(* PLC project bottling_line, Dassault Systèmes ControlBuild 2020 *)
(* stored: creationDateTime 2019-04-23T11:17:34-01:00 *)

CONFIGURATION bottling_line
  VAR_GLOBAL
    generalPanel/acknowledgePB AT 10 : BOOL := false;
    generalPanel/powerUpPB AT 6 : BOOL := false;
    generalPanel/emergencyStopPB AT 7 : BOOL := false;
    generalPanel/manual AT 8 : BOOL := false;
    generalPanel/auto AT 9 : BOOL := false;
    generalPanel/startCyclePB AT 17 : BOOL := false;
    generalPanel/initPB AT 18 : BOOL := false;
    generalPanel/preparationPB AT 19 : BOOL := false;
    generalPanel/productionPB AT 20 : BOOL := false;
    generalPanel/closingPB AT 21 : BOOL := false;
    generalPanel/acknowledgePB/PB AT 10 : BOOL := false;
    generalPanel/acknowledgePB/action AT 39 : BOOL := false;
    generalPanel/acknowledgePB/timeCounter AT 24 : REAL := 0.0;
    generalPanel/acknowledgePB/pulseDuration AT 25 : REAL := 5.0;
    generalPanel/acknowledgePB/PBLogic AT 40 : BOOL := true;
    generalPanel/powerUpPB/PB AT 6 : BOOL := false;
    generalPanel/powerUpPB/action AT 41 : BOOL := false;
    generalPanel/powerUpPB/timeCounter AT 26 : REAL := 0.0;
    generalPanel/powerUpPB/pulseDuration AT 27 : REAL := 5.0;
    generalPanel/powerUpPB/PBLogic AT 42 : BOOL := true;
    generalPanel/emergencyStopPB/pb AT 7 : BOOL := false;
    generalPanel/emergencyStopPB/action AT 43 : BOOL := false;
    generalPanel/emergencyStopPB/PBLogic AT 44 : BOOL := false;
    generalPanel/modesSwitch/leftVariable AT 9 : BOOL := true;
    generalPanel/modesSwitch/rightVariable AT 8 : BOOL := false;
    generalPanel/modesSwitch/leftPosition AT 45 : BOOL := false;
    generalPanel/modesSwitch/rightPosition AT 46 : BOOL := false;
    generalPanel/startCyclePB/PB AT 17 : BOOL := false;
    generalPanel/startCyclePB/action AT 47 : BOOL := false;
    generalPanel/startCyclePB/timeCounter AT 28 : REAL := 0.0;
    generalPanel/startCyclePB/pulseDuration AT 29 : REAL := 5.0;
    generalPanel/startCyclePB/PBLogic AT 48 : BOOL := true;
    generalPanel/initPB/PB AT 18 : BOOL := false;
    generalPanel/initPB/action AT 49 : BOOL := false;
    generalPanel/initPB/timeCounter AT 30 : REAL := 0.0;
    generalPanel/initPB/pulseDuration AT 31 : REAL := 5.0;
    generalPanel/initPB/PBLogic AT 50 : BOOL := true;
    generalPanel/productionSwitch/leftVariable AT 19 : BOOL := true;
    generalPanel/productionSwitch/rightVariable AT 20 : BOOL := false;
    generalPanel/productionSwitch/leftPosition AT 51 : BOOL := false;
    generalPanel/productionSwitch/rightPosition AT 52 : BOOL := false;
    generalPanel/closingPB/PB AT 21 : BOOL := false;
    generalPanel/closingPB/action AT 53 : BOOL := false;
    generalPanel/closingPB/timeCounter AT 32 : REAL := 0.0;
    generalPanel/closingPB/pulseDuration AT 33 : REAL := 5.0;
    generalPanel/closingPB/PBLogic AT 54 : BOOL := true;
    workingModes/powerUpPB AT 6 : BOOL := false;
    workingModes/emergencyStopPB AT 7 : BOOL := false;
    workingModes/manual AT 8 : BOOL := false;
    workingModes/auto AT 9 : BOOL := false;
    workingModes/acknowledgePB AT 10 : BOOL := false;
    workingModes/powerUp AT 5 : BOOL := false;
    workingModes/autoMode AT 28 : BOOL := false;
    workingModes/manualMode AT 29 : BOOL := false;
    workingModes/emStp AT 55 : BOOL := false;
    process/highLevel1 AT 11 : BOOL := false;
    process/lowLevel1 AT 12 : BOOL := false;
    process/highLevel2 AT 13 : BOOL := false;
    process/lowLevel2 AT 14 : BOOL := false;
    process/highLevel3 AT 15 : BOOL := false;
    process/lowLevel3 AT 16 : BOOL := false;
    process/startCyclePB AT 17 : BOOL := false;
    process/initPB AT 18 : BOOL := false;
    process/preparationPB AT 19 : BOOL := false;
    process/productionPB AT 20 : BOOL := false;
    process/closingPB AT 21 : BOOL := false;
    process/pulseGenerator AT 22 : BOOL := false;
    process/bottleFilled AT 23 : BOOL := false;
    process/bottlePresent AT 24 : BOOL := false;
    process/load AT 36 : BOOL := false;
    process/evacuate AT 37 : BOOL := false;
    process/convoy AT 38 : BOOL := false;
    process/pump1 AT 27 : BOOL := false;
    process/pump2 AT 32 : BOOL := false;
    process/valve1 AT 25 : BOOL := false;
    process/valve2 AT 30 : BOOL := false;
    process/valve3 AT 26 : BOOL := false;
    process/valve4 AT 31 : BOOL := false;
    process/loSpeedAgitator AT 35 : BOOL := false;
    process/hiSpeedAgitator AT 34 : BOOL := false;
    process/valve5 AT 33 : BOOL := false;
    process/master/startCyclePB AT 17 : BOOL := false;
    process/master/initPB AT 18 : BOOL := false;
    process/master/preparationPB AT 19 : BOOL := false;
    process/master/productionPB AT 20 : BOOL := false;
    process/master/closingPB AT 21 : BOOL := false;
    process/master/initEnd AT 60 : BOOL := false;
    process/master/preparationEnd AT 61 : BOOL := false;
    process/master/closingEnd AT 62 : BOOL := false;
    process/master/lowLevel3 AT 16 : BOOL := false;
    process/master/initializationRqst AT 59 : BOOL := false;
    process/master/preparationRqst AT 66 : BOOL := false;
    process/master/productionRqst AT 63 : BOOL := false;
    process/master/closingRqst AT 64 : BOOL := false;
    process/master/masterInStandBy AT 65 : BOOL := false;
    process/master/productionWaiting AT 67 : BOOL := false;
    process/master/_X_10 AT 84 : BOOL := true;
    process/master/_X_11 AT 85 : BOOL := false;
    process/master/_X_12 AT 83 : BOOL := false;
    process/master/_X_13 AT 86 : BOOL := false;
    process/master/_X_16 AT 89 : BOOL := false;
    process/master/_X_14 AT 87 : BOOL := false;
    process/master/_X_15 AT 88 : BOOL := false;
    process/tanks/productionRequest AT 63 : BOOL := false;
    process/tanks/closingRequest AT 64 : BOOL := false;
    process/tanks/masterInStandBy AT 65 : BOOL := false;
    process/tanks/highLevel1 AT 11 : BOOL := false;
    process/tanks/highLevel2 AT 13 : BOOL := false;
    process/tanks/highLevel3 AT 15 : BOOL := false;
    process/tanks/lowLevel1 AT 12 : BOOL := false;
    process/tanks/lowLevel2 AT 14 : BOOL := false;
    process/tanks/lowLevel3 AT 16 : BOOL := false;
    process/tanks/pump1 AT 75 : BOOL := false;
    process/tanks/pump2 AT 76 : BOOL := false;
    process/tanks/valve1 AT 77 : BOOL := false;
    process/tanks/valve2 AT 78 : BOOL := false;
    process/tanks/valve3 AT 79 : BOOL := false;
    process/tanks/valve4 AT 80 : BOOL := false;
    process/tanks/lowSpeedAgitator AT 81 : BOOL := false;
    process/tanks/highSpeedAgitator AT 82 : BOOL := false;
    process/tanks/closingEnd AT 62 : BOOL := false;
    process/tanks/_X_10 AT 96 : BOOL := true;
    process/tanks/_X_11 AT 97 : BOOL := false;
    process/tanks/_X_12 AT 98 : BOOL := false;
    process/tanks/_X_13 AT 99 : BOOL := false;
    process/tanks/_X_20 AT 100 : BOOL := true;
    process/tanks/_X_21 AT 101 : BOOL := false;
    process/tanks/_X_30 AT 102 : BOOL := true;
    process/tanks/_X_31 AT 103 : BOOL := false;
    process/preparation/preparationRequest AT 66 : BOOL := false;
    process/preparation/productionWaiting AT 67 : BOOL := false;
    process/preparation/highLevel1 AT 11 : BOOL := false;
    process/preparation/highLevel2 AT 13 : BOOL := false;
    process/preparation/highLevel3 AT 15 : BOOL := false;
    process/preparation/preparationValve1 AT 68 : BOOL := false;
    process/preparation/preparationValve2 AT 69 : BOOL := false;
    process/preparation/preparationValve3 AT 70 : BOOL := false;
    process/preparation/preparationValve4 AT 71 : BOOL := false;
    process/preparation/preparationPump1 AT 72 : BOOL := false;
    process/preparation/preparationPump2 AT 73 : BOOL := false;
    process/preparation/preparationAgit AT 74 : BOOL := false;
    process/preparation/preparationEnd AT 61 : BOOL := false;
    process/preparation/_X_10 AT 109 : BOOL := true;
    process/preparation/_X_11 AT 110 : BOOL := false;
    process/preparation/_X_12 AT 111 : BOOL := false;
    process/preparation/_X_13 AT 112 : BOOL := false;
    process/conveyor/productionRequest AT 63 : BOOL := false;
    process/conveyor/pulseGenerator AT 22 : BOOL := false;
    process/conveyor/bottleFilled AT 23 : BOOL := false;
    process/conveyor/bottlePresent AT 24 : BOOL := false;
    process/conveyor/load AT 36 : BOOL := false;
    process/conveyor/evacuate AT 37 : BOOL := false;
    process/conveyor/convoy AT 38 : BOOL := false;
    process/conveyor/valve5 AT 33 : BOOL := false;
    process/conveyor/encoder AT 528 : INT := 0;
    process/conveyor/_X_10 AT 116 : BOOL := true;
    process/conveyor/_X_11 AT 117 : BOOL := false;
    process/conveyor/_X_12 AT 118 : BOOL := false;
    process/conveyor/_X_13 AT 119 : BOOL := false;
    process/conveyor/_X_14 AT 120 : BOOL := false;
    process/conveyor/value AT 529 : INT := 10;
    process/conveyor/increment AT 530 : INT := 1;
    process/manageFunctionalRq/preparationValve1 AT 68 : BOOL := false;
    process/manageFunctionalRq/preparationValve2 AT 69 : BOOL := false;
    process/manageFunctionalRq/preparationValve3 AT 70 : BOOL := false;
    process/manageFunctionalRq/preparationValve4 AT 71 : BOOL := false;
    process/manageFunctionalRq/preparationPump1 AT 72 : BOOL := false;
    process/manageFunctionalRq/preparationPump2 AT 73 : BOOL := false;
    process/manageFunctionalRq/preparationAgitator AT 74 : BOOL := false;
    process/manageFunctionalRq/productionPump1 AT 75 : BOOL := false;
    process/manageFunctionalRq/productionPump2 AT 76 : BOOL := false;
    process/manageFunctionalRq/productionValve1 AT 77 : BOOL := false;
    process/manageFunctionalRq/productionValve2 AT 78 : BOOL := false;
    process/manageFunctionalRq/productionValve3 AT 79 : BOOL := false;
    process/manageFunctionalRq/productionValve4 AT 80 : BOOL := false;
    process/manageFunctionalRq/productionLSAgitator AT 81 : BOOL := false;
    process/manageFunctionalRq/productionHSAgitator AT 82 : BOOL := false;
    process/manageFunctionalRq/pump1 AT 27 : BOOL := false;
    process/manageFunctionalRq/pump2 AT 32 : BOOL := false;
    process/manageFunctionalRq/valve1 AT 25 : BOOL := false;
    process/manageFunctionalRq/valve2 AT 30 : BOOL := false;
    process/manageFunctionalRq/valve3 AT 26 : BOOL := false;
    process/manageFunctionalRq/valve4 AT 31 : BOOL := false;
    process/manageFunctionalRq/loSpeedAgit AT 35 : BOOL := false;
    process/manageFunctionalRq/hiSpeedAgit AT 34 : BOOL := false;
    pumpingTank1/fillingValve AT 25 : BOOL := false;
    pumpingTank1/emptyingValve AT 26 : BOOL := false;
    pumpingTank1/extractionPump AT 27 : BOOL := false;
    pumpingTank1/acknowledgePB AT 10 : BOOL := false;
    pumpingTank1/autoMode AT 28 : BOOL := false;
    pumpingTank1/manualMode AT 29 : BOOL := false;
    pumpingTank1/lowLevel AT 12 : BOOL := false;
    pumpingTank1/highLevel AT 11 : BOOL := false;
    pumpingTank1/pumpingFlow AT 20 : REAL := 0.0;
    pumpingTank1/level AT 19 : REAL := 0.0;
    pumpingTank1/filling/acknowledgePB AT 10 : BOOL := false;
    pumpingTank1/filling/autoMode AT 28 : BOOL := false;
    pumpingTank1/filling/manualMode AT 29 : BOOL := false;
    pumpingTank1/filling/autoOpenCmd AT 25 : BOOL := false;
    pumpingTank1/filling/inputFlow AT 39 : REAL := 1000.0;
    pumpingTank1/filling/openedSensor AT 135 : BOOL := false;
    pumpingTank1/filling/closedSensor AT 134 : BOOL := false;
    pumpingTank1/filling/generalFault AT 133 : BOOL := false;
    pumpingTank1/filling/outputFlow AT 41 : REAL := 0.0;
    pumpingTank1/filling/percentOpening AT 38 : REAL := 0.0;
    pumpingTank1/filling/panel1/openValvePB AT 139 : BOOL := false;
    pumpingTank1/filling/panel1/switch/variable AT 139 : BOOL := false;
    pumpingTank1/filling/panel1/switch/leftPosition AT 141 : BOOL := false;
    pumpingTank1/filling/panel1/switch/rightPosition AT 142 : BOOL := false;
    pumpingTank1/filling/cmdOfValve/autoMode AT 28 : BOOL := false;
    pumpingTank1/filling/cmdOfValve/manualMode AT 29 : BOOL := false;
    pumpingTank1/filling/cmdOfValve/autoOpenCmd AT 25 : BOOL := false;
    pumpingTank1/filling/cmdOfValve/openValvePB AT 139 : BOOL := false;
    pumpingTank1/filling/cmdOfValve/openedSensorFB AT 135 : BOOL := false;
    pumpingTank1/filling/cmdOfValve/closedSensorFB AT 134 : BOOL := false;
    pumpingTank1/filling/cmdOfValve/acknowledgePB AT 10 : BOOL := false;
    pumpingTank1/filling/cmdOfValve/openCmd AT 140 : BOOL := false;
    pumpingTank1/filling/cmdOfValve/generalFault AT 133 : BOOL := false;
    pumpingTank1/filling/cmdOfValve/actions/autoMode AT 28 : BOOL := false;
    pumpingTank1/filling/cmdOfValve/actions/manualMode AT 29 : BOOL := false;
    pumpingTank1/filling/cmdOfValve/actions/autoOpenCmd AT 25 : BOOL := false;
    pumpingTank1/filling/cmdOfValve/actions/openValvePB AT 139 : BOOL := false;
    pumpingTank1/filling/cmdOfValve/actions/generalFault AT 133 : BOOL := false;
    pumpingTank1/filling/cmdOfValve/actions/openCmd AT 140 : BOOL := false;
    pumpingTank1/filling/cmdOfValve/faults1/openCmd AT 140 : BOOL := false;
    pumpingTank1/filling/cmdOfValve/faults1/openedSensorFB AT 135 : BOOL := false;
    pumpingTank1/filling/cmdOfValve/faults1/closedSensorFB AT 134 : BOOL := false;
    pumpingTank1/filling/cmdOfValve/faults1/acknowledgePB AT 10 : BOOL := false;
    pumpingTank1/filling/cmdOfValve/faults1/generalFault AT 133 : BOOL := false;
    pumpingTank1/filling/cmdOfValve/faults1/discordanceFault AT 143 : BOOL := false;
    pumpingTank1/filling/cmdOfValve/faults1/openedSensorFault AT 144 : BOOL := false;
    pumpingTank1/filling/cmdOfValve/faults1/closedSensorFault AT 145 : BOOL := false;
    pumpingTank1/filling/cmdOfValve/faults1/presetMvt AT 536 : TIME := T#0h0m4s0ms;
    pumpingTank1/filling/cmdOfValve/faults1/presetDiscordance AT 540 : TIME := T#0h0m0s200ms;
    pumpingTank1/filling/valve/voltage380 AT 138 : BOOL := true;
    pumpingTank1/filling/valve/cmdSupply AT 137 : BOOL := true;
    pumpingTank1/filling/valve/sensorSupply AT 136 : BOOL := true;
    pumpingTank1/filling/valve/openCmd AT 140 : BOOL := false;
    pumpingTank1/filling/valve/inputFlow AT 39 : REAL := 1000.0;
    pumpingTank1/filling/valve/openedSensor AT 135 : BOOL := false;
    pumpingTank1/filling/valve/closedSensor AT 134 : BOOL := false;
    pumpingTank1/filling/valve/outputFlow AT 41 : REAL := 0.0;
    pumpingTank1/filling/valve/percentOpening AT 38 : REAL := 0.0;
    pumpingTank1/filling/valve/increment AT 44 : REAL := 0.0;
    pumpingTank1/filling/valve/openState AT 152 : BOOL := false;
    pumpingTank1/filling/valve/closeState AT 153 : BOOL := false;
    pumpingTank1/filling/valve/openingVal AT 45 : REAL := 0.0;
    pumpingTank1/filling/valve/unit AT 46 : REAL := 0.0;
    pumpingTank1/filling/valve/openingTime AT 47 : REAL := 2.0;
    pumpingTank1/filling/valve/openedSensorLogic AT 154 : BOOL := true;
    pumpingTank1/filling/valve/closedSensorLogic AT 155 : BOOL := true;
    pumpingTank1/filling/valve/flowMax AT 48 : REAL := 1000.0;
    pumpingTank1/filling/valve/flowPerHour AT 156 : BOOL := false;
    pumpingTank1/filling/valve/flowPerMinute AT 157 : BOOL := true;
    pumpingTank1/filling/valve/d_locking AT 158 : BOOL := false;
    pumpingTank1/filling/valve/v_d_locking AT 49 : REAL := 0.0;
    pumpingTank1/filling/valve/d_flow AT 159 : BOOL := false;
    pumpingTank1/filling/valve/v_d_flow AT 50 : REAL := 0.0;
    pumpingTank1/filling/valve/d_electrical AT 160 : BOOL := false;
    pumpingTank1/filling/valve/v_d_electrical AT 161 : BOOL := false;
    pumpingTank1/filling/valve/d_openedSensor AT 162 : BOOL := false;
    pumpingTank1/filling/valve/v_d_openedSensor AT 163 : BOOL := false;
    pumpingTank1/filling/valve/d_closedSensor AT 164 : BOOL := false;
    pumpingTank1/filling/valve/v_d_closedSensor AT 165 : BOOL := false;
    pumpingTank1/emptying/acknowledgePB AT 10 : BOOL := false;
    pumpingTank1/emptying/autoMode AT 28 : BOOL := false;
    pumpingTank1/emptying/manualMode AT 29 : BOOL := false;
    pumpingTank1/emptying/autoOpenCmd AT 26 : BOOL := false;
    pumpingTank1/emptying/inputFlow AT 40 : REAL := 0.0;
    pumpingTank1/emptying/openedSensor AT 132 : BOOL := false;
    pumpingTank1/emptying/closedSensor AT 131 : BOOL := false;
    pumpingTank1/emptying/generalFault AT 130 : BOOL := false;
    pumpingTank1/emptying/outputFlow AT 20 : REAL := 0.0;
    pumpingTank1/emptying/percentOpening AT 37 : REAL := 0.0;
    pumpingTank1/emptying/panel1/openValvePB AT 169 : BOOL := false;
    pumpingTank1/emptying/panel1/switch/variable AT 169 : BOOL := false;
    pumpingTank1/emptying/panel1/switch/leftPosition AT 171 : BOOL := false;
    pumpingTank1/emptying/panel1/switch/rightPosition AT 172 : BOOL := false;
    pumpingTank1/emptying/cmdOfValve/autoMode AT 28 : BOOL := false;
    pumpingTank1/emptying/cmdOfValve/manualMode AT 29 : BOOL := false;
    pumpingTank1/emptying/cmdOfValve/autoOpenCmd AT 26 : BOOL := false;
    pumpingTank1/emptying/cmdOfValve/openValvePB AT 169 : BOOL := false;
    pumpingTank1/emptying/cmdOfValve/openedSensorFB AT 132 : BOOL := false;
    pumpingTank1/emptying/cmdOfValve/closedSensorFB AT 131 : BOOL := false;
    pumpingTank1/emptying/cmdOfValve/acknowledgePB AT 10 : BOOL := false;
    pumpingTank1/emptying/cmdOfValve/openCmd AT 170 : BOOL := false;
    pumpingTank1/emptying/cmdOfValve/generalFault AT 130 : BOOL := false;
    pumpingTank1/emptying/cmdOfValve/actions/autoMode AT 28 : BOOL := false;
    pumpingTank1/emptying/cmdOfValve/actions/manualMode AT 29 : BOOL := false;
    pumpingTank1/emptying/cmdOfValve/actions/autoOpenCmd AT 26 : BOOL := false;
    pumpingTank1/emptying/cmdOfValve/actions/openValvePB AT 169 : BOOL := false;
    pumpingTank1/emptying/cmdOfValve/actions/generalFault AT 130 : BOOL := false;
    pumpingTank1/emptying/cmdOfValve/actions/openCmd AT 170 : BOOL := false;
    pumpingTank1/emptying/cmdOfValve/faults1/openCmd AT 170 : BOOL := false;
    pumpingTank1/emptying/cmdOfValve/faults1/openedSensorFB AT 132 : BOOL := false;
    pumpingTank1/emptying/cmdOfValve/faults1/closedSensorFB AT 131 : BOOL := false;
    pumpingTank1/emptying/cmdOfValve/faults1/acknowledgePB AT 10 : BOOL := false;
    pumpingTank1/emptying/cmdOfValve/faults1/generalFault AT 130 : BOOL := false;
    pumpingTank1/emptying/cmdOfValve/faults1/discordanceFault AT 173 : BOOL := false;
    pumpingTank1/emptying/cmdOfValve/faults1/openedSensorFault AT 174 : BOOL := false;
    pumpingTank1/emptying/cmdOfValve/faults1/closedSensorFault AT 175 : BOOL := false;
    pumpingTank1/emptying/cmdOfValve/faults1/presetMvt AT 568 : TIME := T#0h0m4s0ms;
    pumpingTank1/emptying/cmdOfValve/faults1/presetDiscordance AT 572 : TIME := T#0h0m0s200ms;
    pumpingTank1/emptying/valve/voltage380 AT 168 : BOOL := true;
    pumpingTank1/emptying/valve/cmdSupply AT 167 : BOOL := true;
    pumpingTank1/emptying/valve/sensorSupply AT 166 : BOOL := true;
    pumpingTank1/emptying/valve/openCmd AT 170 : BOOL := false;
    pumpingTank1/emptying/valve/inputFlow AT 40 : REAL := 0.0;
    pumpingTank1/emptying/valve/openedSensor AT 132 : BOOL := false;
    pumpingTank1/emptying/valve/closedSensor AT 131 : BOOL := false;
    pumpingTank1/emptying/valve/outputFlow AT 20 : REAL := 0.0;
    pumpingTank1/emptying/valve/percentOpening AT 37 : REAL := 0.0;
    pumpingTank1/emptying/valve/increment AT 51 : REAL := 0.0;
    pumpingTank1/emptying/valve/openState AT 182 : BOOL := false;
    pumpingTank1/emptying/valve/closeState AT 183 : BOOL := false;
    pumpingTank1/emptying/valve/openingVal AT 52 : REAL := 0.0;
    pumpingTank1/emptying/valve/unit AT 53 : REAL := 0.0;
    pumpingTank1/emptying/valve/openingTime AT 54 : REAL := 2.0;
    pumpingTank1/emptying/valve/openedSensorLogic AT 184 : BOOL := true;
    pumpingTank1/emptying/valve/closedSensorLogic AT 185 : BOOL := true;
    pumpingTank1/emptying/valve/flowMax AT 55 : REAL := 1000.0;
    pumpingTank1/emptying/valve/flowPerHour AT 186 : BOOL := false;
    pumpingTank1/emptying/valve/flowPerMinute AT 187 : BOOL := true;
    pumpingTank1/emptying/valve/d_locking AT 188 : BOOL := false;
    pumpingTank1/emptying/valve/v_d_locking AT 56 : REAL := 0.0;
    pumpingTank1/emptying/valve/d_flow AT 189 : BOOL := false;
    pumpingTank1/emptying/valve/v_d_flow AT 57 : REAL := 0.0;
    pumpingTank1/emptying/valve/d_electrical AT 190 : BOOL := false;
    pumpingTank1/emptying/valve/v_d_electrical AT 191 : BOOL := false;
    pumpingTank1/emptying/valve/d_openedSensor AT 192 : BOOL := false;
    pumpingTank1/emptying/valve/v_d_openedSensor AT 193 : BOOL := false;
    pumpingTank1/emptying/valve/d_closedSensor AT 194 : BOOL := false;
    pumpingTank1/emptying/valve/v_d_closedSensor AT 195 : BOOL := false;
    pumpingTank1/tank/inletFlow AT 41 : REAL := 0.0;
    pumpingTank1/tank/outletFlow AT 20 : REAL := 0.0;
    pumpingTank1/tank/tankLevel AT 42 : REAL := 0.0;
    pumpingTank1/tank/percent AT 58 : REAL := 0.0;
    pumpingTank1/tank/capacity AT 59 : REAL := 500.0;
    pumpingTank1/tank/d_level AT 196 : BOOL := false;
    pumpingTank1/tank/v_d_level AT 60 : REAL := 0.0;
    pumpingTank1/extraction/acknowledgePB AT 10 : BOOL := false;
    pumpingTank1/extraction/autoMode AT 28 : BOOL := false;
    pumpingTank1/extraction/manualMode AT 29 : BOOL := false;
    pumpingTank1/extraction/autoCmd AT 27 : BOOL := false;
    pumpingTank1/extraction/inputFlow AT 42 : REAL := 0.0;
    pumpingTank1/extraction/generalFault AT 129 : BOOL := false;
    pumpingTank1/extraction/speedVal AT 36 : REAL := 0.0;
    pumpingTank1/extraction/outputFlow AT 40 : REAL := 0.0;
    pumpingTank1/extraction/panel1/onPB AT 203 : BOOL := false;
    pumpingTank1/extraction/panel1/offPB AT 204 : BOOL := false;
    pumpingTank1/extraction/panel1/onPB/PB AT 203 : BOOL := false;
    pumpingTank1/extraction/panel1/onPB/action AT 205 : BOOL := false;
    pumpingTank1/extraction/panel1/onPB/timeCounter AT 61 : REAL := 0.0;
    pumpingTank1/extraction/panel1/onPB/pulseDuration AT 62 : REAL := 5.0;
    pumpingTank1/extraction/panel1/onPB/PBLogic AT 206 : BOOL := true;
    pumpingTank1/extraction/panel1/offPB/PB AT 204 : BOOL := false;
    pumpingTank1/extraction/panel1/offPB/action AT 207 : BOOL := false;
    pumpingTank1/extraction/panel1/offPB/timeCounter AT 63 : REAL := 0.0;
    pumpingTank1/extraction/panel1/offPB/pulseDuration AT 64 : REAL := 5.0;
    pumpingTank1/extraction/panel1/offPB/PBLogic AT 208 : BOOL := true;
    pumpingTank1/extraction/pump/voltage380 AT 199 : BOOL := true;
    pumpingTank1/extraction/pump/cmdSupply AT 198 : BOOL := true;
    pumpingTank1/extraction/pump/sensorSupply AT 197 : BOOL := true;
    pumpingTank1/extraction/pump/onCmd AT 200 : BOOL := false;
    pumpingTank1/extraction/pump/inputFlow AT 42 : REAL := 0.0;
    pumpingTank1/extraction/pump/onFB AT 202 : BOOL := false;
    pumpingTank1/extraction/pump/thermal AT 201 : BOOL := false;
    pumpingTank1/extraction/pump/speedVal AT 36 : REAL := 0.0;
    pumpingTank1/extraction/pump/outputFlow AT 40 : REAL := 0.0;
    pumpingTank1/extraction/pump/increment AT 65 : REAL := 0.0;
    pumpingTank1/extraction/pump/onState AT 209 : BOOL := false;
    pumpingTank1/extraction/pump/speedSetpoint AT 66 : REAL := 0.0;
    pumpingTank1/extraction/pump/unit AT 67 : REAL := 0.0;
    pumpingTank1/extraction/pump/nominalTime AT 68 : REAL := 2.0;
    pumpingTank1/extraction/pump/thermalLogic AT 210 : BOOL := false;
    pumpingTank1/extraction/pump/onFbLogic AT 211 : BOOL := true;
    pumpingTank1/extraction/pump/flowMax AT 69 : REAL := 1000.0;
    pumpingTank1/extraction/pump/nominalSpeed AT 70 : REAL := 3600.0;
    pumpingTank1/extraction/pump/flowPerHour AT 212 : BOOL := false;
    pumpingTank1/extraction/pump/flowPerMinute AT 213 : BOOL := true;
    pumpingTank1/extraction/pump/d_locking AT 214 : BOOL := false;
    pumpingTank1/extraction/pump/v_d_locking AT 71 : REAL := 0.0;
    pumpingTank1/extraction/pump/d_flow AT 215 : BOOL := false;
    pumpingTank1/extraction/pump/v_d_flow AT 72 : REAL := 0.0;
    pumpingTank1/extraction/pump/d_electrical AT 216 : BOOL := false;
    pumpingTank1/extraction/pump/v_d_electrical AT 217 : BOOL := false;
    pumpingTank1/extraction/pump/d_onFB AT 218 : BOOL := false;
    pumpingTank1/extraction/pump/v_d_onFB AT 219 : BOOL := false;
    pumpingTank1/extraction/cmdOfMotor/autoMode AT 28 : BOOL := false;
    pumpingTank1/extraction/cmdOfMotor/manualMode AT 29 : BOOL := false;
    pumpingTank1/extraction/cmdOfMotor/autoCmd AT 27 : BOOL := false;
    pumpingTank1/extraction/cmdOfMotor/thermalFB AT 201 : BOOL := false;
    pumpingTank1/extraction/cmdOfMotor/onFB AT 202 : BOOL := false;
    pumpingTank1/extraction/cmdOfMotor/onPB AT 203 : BOOL := false;
    pumpingTank1/extraction/cmdOfMotor/offPB AT 204 : BOOL := false;
    pumpingTank1/extraction/cmdOfMotor/acknowledgePB AT 10 : BOOL := false;
    pumpingTank1/extraction/cmdOfMotor/cmd AT 200 : BOOL := false;
    pumpingTank1/extraction/cmdOfMotor/generalFault AT 129 : BOOL := false;
    pumpingTank1/extraction/cmdOfMotor/actions/autoMode AT 28 : BOOL := false;
    pumpingTank1/extraction/cmdOfMotor/actions/manualMode AT 29 : BOOL := false;
    pumpingTank1/extraction/cmdOfMotor/actions/autoCmd AT 27 : BOOL := false;
    pumpingTank1/extraction/cmdOfMotor/actions/onPB AT 203 : BOOL := false;
    pumpingTank1/extraction/cmdOfMotor/actions/offPB AT 204 : BOOL := false;
    pumpingTank1/extraction/cmdOfMotor/actions/generalFault AT 129 : BOOL := false;
    pumpingTank1/extraction/cmdOfMotor/actions/cmd AT 200 : BOOL := false;
    pumpingTank1/extraction/cmdOfMotor/faults1/cmd AT 200 : BOOL := false;
    pumpingTank1/extraction/cmdOfMotor/faults1/thermalFB AT 201 : BOOL := false;
    pumpingTank1/extraction/cmdOfMotor/faults1/onFB AT 202 : BOOL := false;
    pumpingTank1/extraction/cmdOfMotor/faults1/acknowledgePB AT 10 : BOOL := false;
    pumpingTank1/extraction/cmdOfMotor/faults1/generalFault AT 129 : BOOL := false;
    pumpingTank1/extraction/cmdOfMotor/faults1/thermalFault AT 220 : BOOL := false;
    pumpingTank1/extraction/cmdOfMotor/faults1/onFBFault AT 221 : BOOL := false;
    pumpingTank1/levelScale/inputValue AT 42 : REAL := 0.0;
    pumpingTank1/levelScale/realValue AT 43 : REAL := 0.0;
    pumpingTank1/levelScale/dintValue AT 535 : DINT := 0;
    pumpingTank1/levelScale/intValue AT 534 : INT := 0;
    pumpingTank1/levelScale/a AT 73 : REAL := 0.0;
    pumpingTank1/levelScale/b AT 74 : REAL := 0.0;
    pumpingTank1/levelScale/k AT 75 : REAL := 0.0;
    pumpingTank1/levelScale/minInput AT 76 : REAL := 0.0;
    pumpingTank1/levelScale/maxInput AT 77 : REAL := 500.0;
    pumpingTank1/levelScale/minOutput AT 78 : REAL := 0.0;
    pumpingTank1/levelScale/maxOutput AT 79 : REAL := 100.0;
    pumpingTank1/levelScale/d_scale AT 224 : BOOL := false;
    pumpingTank1/levelScale/v_d_scale AT 80 : REAL := 0.0;
    pumpingTank1/highLevel/level AT 42 : REAL := 0.0;
    pumpingTank1/highLevel/sensorSupply AT 128 : BOOL := true;
    pumpingTank1/highLevel/thresholdSensor AT 11 : BOOL := false;
    pumpingTank1/highLevel/threshold AT 81 : REAL := 490.0;
    pumpingTank1/highLevel/wiringLogic AT 225 : BOOL := true;
    pumpingTank1/highLevel/d_sensor AT 226 : BOOL := false;
    pumpingTank1/highLevel/v_d_sensor AT 227 : BOOL := false;
    pumpingTank1/lowLevel/level AT 42 : REAL := 0.0;
    pumpingTank1/lowLevel/sensorSupply AT 127 : BOOL := true;
    pumpingTank1/lowLevel/thresholdSensor AT 12 : BOOL := false;
    pumpingTank1/lowLevel/threshold AT 82 : REAL := 30.0;
    pumpingTank1/lowLevel/wiringLogic AT 228 : BOOL := false;
    pumpingTank1/lowLevel/d_sensor AT 229 : BOOL := false;
    pumpingTank1/lowLevel/v_d_sensor AT 230 : BOOL := false;
    pumpingTank1/levelMeasurement/measure AT 43 : REAL := 0.0;
    pumpingTank1/levelMeasurement/sensorSupply AT 126 : BOOL := true;
    pumpingTank1/levelMeasurement/realValue AT 19 : REAL := 0.0;
    pumpingTank1/levelMeasurement/intValue AT 35 : REAL := 0.0;
    pumpingTank1/levelMeasurement/dintValue AT 34 : REAL := 0.0;
    pumpingTank1/levelMeasurement/tmp AT 608 : DINT := 0;
    pumpingTank1/levelMeasurement/localValue AT 83 : REAL := 0.0;
    pumpingTank1/levelMeasurement/nbDigit AT 609 : SINT := 2;
    pumpingTank1/levelMeasurement/d_value AT 231 : BOOL := false;
    pumpingTank1/levelMeasurement/v_d_value AT 84 : REAL := 0.0;
    pumpingTank2/fillingValve AT 30 : BOOL := false;
    pumpingTank2/emptyingValve AT 31 : BOOL := false;
    pumpingTank2/extractionPump AT 32 : BOOL := false;
    pumpingTank2/acknowledgePB AT 10 : BOOL := false;
    pumpingTank2/autoMode AT 28 : BOOL := false;
    pumpingTank2/manualMode AT 29 : BOOL := false;
    pumpingTank2/lowLevel AT 14 : BOOL := false;
    pumpingTank2/highLevel AT 13 : BOOL := false;
    pumpingTank2/pumpingFlow AT 21 : REAL := 0.0;
    pumpingTank2/level AT 18 : REAL := 0.0;
    pumpingTank2/filling/acknowledgePB AT 10 : BOOL := false;
    pumpingTank2/filling/autoMode AT 28 : BOOL := false;
    pumpingTank2/filling/manualMode AT 29 : BOOL := false;
    pumpingTank2/filling/autoOpenCmd AT 30 : BOOL := false;
    pumpingTank2/filling/inputFlow AT 90 : REAL := 1000.0;
    pumpingTank2/filling/openedSensor AT 241 : BOOL := false;
    pumpingTank2/filling/closedSensor AT 240 : BOOL := false;
    pumpingTank2/filling/generalFault AT 239 : BOOL := false;
    pumpingTank2/filling/outputFlow AT 92 : REAL := 0.0;
    pumpingTank2/filling/percentOpening AT 89 : REAL := 0.0;
    pumpingTank2/filling/panel1/openValvePB AT 245 : BOOL := false;
    pumpingTank2/filling/panel1/switch/variable AT 245 : BOOL := false;
    pumpingTank2/filling/panel1/switch/leftPosition AT 247 : BOOL := false;
    pumpingTank2/filling/panel1/switch/rightPosition AT 248 : BOOL := false;
    pumpingTank2/filling/cmdOfValve/autoMode AT 28 : BOOL := false;
    pumpingTank2/filling/cmdOfValve/manualMode AT 29 : BOOL := false;
    pumpingTank2/filling/cmdOfValve/autoOpenCmd AT 30 : BOOL := false;
    pumpingTank2/filling/cmdOfValve/openValvePB AT 245 : BOOL := false;
    pumpingTank2/filling/cmdOfValve/openedSensorFB AT 241 : BOOL := false;
    pumpingTank2/filling/cmdOfValve/closedSensorFB AT 240 : BOOL := false;
    pumpingTank2/filling/cmdOfValve/acknowledgePB AT 10 : BOOL := false;
    pumpingTank2/filling/cmdOfValve/openCmd AT 246 : BOOL := false;
    pumpingTank2/filling/cmdOfValve/generalFault AT 239 : BOOL := false;
    pumpingTank2/filling/cmdOfValve/actions/autoMode AT 28 : BOOL := false;
    pumpingTank2/filling/cmdOfValve/actions/manualMode AT 29 : BOOL := false;
    pumpingTank2/filling/cmdOfValve/actions/autoOpenCmd AT 30 : BOOL := false;
    pumpingTank2/filling/cmdOfValve/actions/openValvePB AT 245 : BOOL := false;
    pumpingTank2/filling/cmdOfValve/actions/generalFault AT 239 : BOOL := false;
    pumpingTank2/filling/cmdOfValve/actions/openCmd AT 246 : BOOL := false;
    pumpingTank2/filling/cmdOfValve/faults1/openCmd AT 246 : BOOL := false;
    pumpingTank2/filling/cmdOfValve/faults1/openedSensorFB AT 241 : BOOL := false;
    pumpingTank2/filling/cmdOfValve/faults1/closedSensorFB AT 240 : BOOL := false;
    pumpingTank2/filling/cmdOfValve/faults1/acknowledgePB AT 10 : BOOL := false;
    pumpingTank2/filling/cmdOfValve/faults1/generalFault AT 239 : BOOL := false;
    pumpingTank2/filling/cmdOfValve/faults1/discordanceFault AT 249 : BOOL := false;
    pumpingTank2/filling/cmdOfValve/faults1/openedSensorFault AT 250 : BOOL := false;
    pumpingTank2/filling/cmdOfValve/faults1/closedSensorFault AT 251 : BOOL := false;
    pumpingTank2/filling/cmdOfValve/faults1/presetMvt AT 612 : TIME := T#0h0m4s0ms;
    pumpingTank2/filling/cmdOfValve/faults1/presetDiscordance AT 616 : TIME := T#0h0m0s200ms;
    pumpingTank2/filling/valve/voltage380 AT 244 : BOOL := true;
    pumpingTank2/filling/valve/cmdSupply AT 243 : BOOL := true;
    pumpingTank2/filling/valve/sensorSupply AT 242 : BOOL := true;
    pumpingTank2/filling/valve/openCmd AT 246 : BOOL := false;
    pumpingTank2/filling/valve/inputFlow AT 90 : REAL := 1000.0;
    pumpingTank2/filling/valve/openedSensor AT 241 : BOOL := false;
    pumpingTank2/filling/valve/closedSensor AT 240 : BOOL := false;
    pumpingTank2/filling/valve/outputFlow AT 92 : REAL := 0.0;
    pumpingTank2/filling/valve/percentOpening AT 89 : REAL := 0.0;
    pumpingTank2/filling/valve/increment AT 95 : REAL := 0.0;
    pumpingTank2/filling/valve/openState AT 258 : BOOL := false;
    pumpingTank2/filling/valve/closeState AT 259 : BOOL := false;
    pumpingTank2/filling/valve/openingVal AT 96 : REAL := 0.0;
    pumpingTank2/filling/valve/unit AT 97 : REAL := 0.0;
    pumpingTank2/filling/valve/openingTime AT 98 : REAL := 2.0;
    pumpingTank2/filling/valve/openedSensorLogic AT 260 : BOOL := true;
    pumpingTank2/filling/valve/closedSensorLogic AT 261 : BOOL := true;
    pumpingTank2/filling/valve/flowMax AT 99 : REAL := 1000.0;
    pumpingTank2/filling/valve/flowPerHour AT 262 : BOOL := false;
    pumpingTank2/filling/valve/flowPerMinute AT 263 : BOOL := true;
    pumpingTank2/filling/valve/d_locking AT 264 : BOOL := false;
    pumpingTank2/filling/valve/v_d_locking AT 100 : REAL := 0.0;
    pumpingTank2/filling/valve/d_flow AT 265 : BOOL := false;
    pumpingTank2/filling/valve/v_d_flow AT 101 : REAL := 0.0;
    pumpingTank2/filling/valve/d_electrical AT 266 : BOOL := false;
    pumpingTank2/filling/valve/v_d_electrical AT 267 : BOOL := false;
    pumpingTank2/filling/valve/d_openedSensor AT 268 : BOOL := false;
    pumpingTank2/filling/valve/v_d_openedSensor AT 269 : BOOL := false;
    pumpingTank2/filling/valve/d_closedSensor AT 270 : BOOL := false;
    pumpingTank2/filling/valve/v_d_closedSensor AT 271 : BOOL := false;
    pumpingTank2/emptying/acknowledgePB AT 10 : BOOL := false;
    pumpingTank2/emptying/autoMode AT 28 : BOOL := false;
    pumpingTank2/emptying/manualMode AT 29 : BOOL := false;
    pumpingTank2/emptying/autoOpenCmd AT 31 : BOOL := false;
    pumpingTank2/emptying/inputFlow AT 91 : REAL := 0.0;
    pumpingTank2/emptying/openedSensor AT 238 : BOOL := false;
    pumpingTank2/emptying/closedSensor AT 237 : BOOL := false;
    pumpingTank2/emptying/generalFault AT 236 : BOOL := false;
    pumpingTank2/emptying/outputFlow AT 21 : REAL := 0.0;
    pumpingTank2/emptying/percentOpening AT 88 : REAL := 0.0;
    pumpingTank2/emptying/panel1/openValvePB AT 275 : BOOL := false;
    pumpingTank2/emptying/panel1/switch/variable AT 275 : BOOL := false;
    pumpingTank2/emptying/panel1/switch/leftPosition AT 277 : BOOL := false;
    pumpingTank2/emptying/panel1/switch/rightPosition AT 278 : BOOL := false;
    pumpingTank2/emptying/cmdOfValve/autoMode AT 28 : BOOL := false;
    pumpingTank2/emptying/cmdOfValve/manualMode AT 29 : BOOL := false;
    pumpingTank2/emptying/cmdOfValve/autoOpenCmd AT 31 : BOOL := false;
    pumpingTank2/emptying/cmdOfValve/openValvePB AT 275 : BOOL := false;
    pumpingTank2/emptying/cmdOfValve/openedSensorFB AT 238 : BOOL := false;
    pumpingTank2/emptying/cmdOfValve/closedSensorFB AT 237 : BOOL := false;
    pumpingTank2/emptying/cmdOfValve/acknowledgePB AT 10 : BOOL := false;
    pumpingTank2/emptying/cmdOfValve/openCmd AT 276 : BOOL := false;
    pumpingTank2/emptying/cmdOfValve/generalFault AT 236 : BOOL := false;
    pumpingTank2/emptying/cmdOfValve/actions/autoMode AT 28 : BOOL := false;
    pumpingTank2/emptying/cmdOfValve/actions/manualMode AT 29 : BOOL := false;
    pumpingTank2/emptying/cmdOfValve/actions/autoOpenCmd AT 31 : BOOL := false;
    pumpingTank2/emptying/cmdOfValve/actions/openValvePB AT 275 : BOOL := false;
    pumpingTank2/emptying/cmdOfValve/actions/generalFault AT 236 : BOOL := false;
    pumpingTank2/emptying/cmdOfValve/actions/openCmd AT 276 : BOOL := false;
    pumpingTank2/emptying/cmdOfValve/faults1/openCmd AT 276 : BOOL := false;
    pumpingTank2/emptying/cmdOfValve/faults1/openedSensorFB AT 238 : BOOL := false;
    pumpingTank2/emptying/cmdOfValve/faults1/closedSensorFB AT 237 : BOOL := false;
    pumpingTank2/emptying/cmdOfValve/faults1/acknowledgePB AT 10 : BOOL := false;
    pumpingTank2/emptying/cmdOfValve/faults1/generalFault AT 236 : BOOL := false;
    pumpingTank2/emptying/cmdOfValve/faults1/discordanceFault AT 279 : BOOL := false;
    pumpingTank2/emptying/cmdOfValve/faults1/openedSensorFault AT 280 : BOOL := false;
    pumpingTank2/emptying/cmdOfValve/faults1/closedSensorFault AT 281 : BOOL := false;
    pumpingTank2/emptying/cmdOfValve/faults1/presetMvt AT 644 : TIME := T#0h0m4s0ms;
    pumpingTank2/emptying/cmdOfValve/faults1/presetDiscordance AT 648 : TIME := T#0h0m0s200ms;
    pumpingTank2/emptying/valve/voltage380 AT 274 : BOOL := true;
    pumpingTank2/emptying/valve/cmdSupply AT 273 : BOOL := true;
    pumpingTank2/emptying/valve/sensorSupply AT 272 : BOOL := true;
    pumpingTank2/emptying/valve/openCmd AT 276 : BOOL := false;
    pumpingTank2/emptying/valve/inputFlow AT 91 : REAL := 0.0;
    pumpingTank2/emptying/valve/openedSensor AT 238 : BOOL := false;
    pumpingTank2/emptying/valve/closedSensor AT 237 : BOOL := false;
    pumpingTank2/emptying/valve/outputFlow AT 21 : REAL := 0.0;
    pumpingTank2/emptying/valve/percentOpening AT 88 : REAL := 0.0;
    pumpingTank2/emptying/valve/increment AT 102 : REAL := 0.0;
    pumpingTank2/emptying/valve/openState AT 288 : BOOL := false;
    pumpingTank2/emptying/valve/closeState AT 289 : BOOL := false;
    pumpingTank2/emptying/valve/openingVal AT 103 : REAL := 0.0;
    pumpingTank2/emptying/valve/unit AT 104 : REAL := 0.0;
    pumpingTank2/emptying/valve/openingTime AT 105 : REAL := 2.0;
    pumpingTank2/emptying/valve/openedSensorLogic AT 290 : BOOL := true;
    pumpingTank2/emptying/valve/closedSensorLogic AT 291 : BOOL := true;
    pumpingTank2/emptying/valve/flowMax AT 106 : REAL := 1000.0;
    pumpingTank2/emptying/valve/flowPerHour AT 292 : BOOL := false;
    pumpingTank2/emptying/valve/flowPerMinute AT 293 : BOOL := true;
    pumpingTank2/emptying/valve/d_locking AT 294 : BOOL := false;
    pumpingTank2/emptying/valve/v_d_locking AT 107 : REAL := 0.0;
    pumpingTank2/emptying/valve/d_flow AT 295 : BOOL := false;
    pumpingTank2/emptying/valve/v_d_flow AT 108 : REAL := 0.0;
    pumpingTank2/emptying/valve/d_electrical AT 296 : BOOL := false;
    pumpingTank2/emptying/valve/v_d_electrical AT 297 : BOOL := false;
    pumpingTank2/emptying/valve/d_openedSensor AT 298 : BOOL := false;
    pumpingTank2/emptying/valve/v_d_openedSensor AT 299 : BOOL := false;
    pumpingTank2/emptying/valve/d_closedSensor AT 300 : BOOL := false;
    pumpingTank2/emptying/valve/v_d_closedSensor AT 301 : BOOL := false;
    pumpingTank2/tank/inletFlow AT 92 : REAL := 0.0;
    pumpingTank2/tank/outletFlow AT 21 : REAL := 0.0;
    pumpingTank2/tank/tankLevel AT 93 : REAL := 0.0;
    pumpingTank2/tank/percent AT 109 : REAL := 0.0;
    pumpingTank2/tank/capacity AT 110 : REAL := 500.0;
    pumpingTank2/tank/d_level AT 302 : BOOL := false;
    pumpingTank2/tank/v_d_level AT 111 : REAL := 0.0;
    pumpingTank2/extraction/acknowledgePB AT 10 : BOOL := false;
    pumpingTank2/extraction/autoMode AT 28 : BOOL := false;
    pumpingTank2/extraction/manualMode AT 29 : BOOL := false;
    pumpingTank2/extraction/autoCmd AT 32 : BOOL := false;
    pumpingTank2/extraction/inputFlow AT 93 : REAL := 0.0;
    pumpingTank2/extraction/generalFault AT 235 : BOOL := false;
    pumpingTank2/extraction/speedVal AT 87 : REAL := 0.0;
    pumpingTank2/extraction/outputFlow AT 91 : REAL := 0.0;
    pumpingTank2/extraction/panel1/onPB AT 309 : BOOL := false;
    pumpingTank2/extraction/panel1/offPB AT 310 : BOOL := false;
    pumpingTank2/extraction/panel1/onPB/PB AT 309 : BOOL := false;
    pumpingTank2/extraction/panel1/onPB/action AT 311 : BOOL := false;
    pumpingTank2/extraction/panel1/onPB/timeCounter AT 112 : REAL := 0.0;
    pumpingTank2/extraction/panel1/onPB/pulseDuration AT 113 : REAL := 5.0;
    pumpingTank2/extraction/panel1/onPB/PBLogic AT 312 : BOOL := true;
    pumpingTank2/extraction/panel1/offPB/PB AT 310 : BOOL := false;
    pumpingTank2/extraction/panel1/offPB/action AT 313 : BOOL := false;
    pumpingTank2/extraction/panel1/offPB/timeCounter AT 114 : REAL := 0.0;
    pumpingTank2/extraction/panel1/offPB/pulseDuration AT 115 : REAL := 5.0;
    pumpingTank2/extraction/panel1/offPB/PBLogic AT 314 : BOOL := true;
    pumpingTank2/extraction/pump/voltage380 AT 305 : BOOL := true;
    pumpingTank2/extraction/pump/cmdSupply AT 304 : BOOL := true;
    pumpingTank2/extraction/pump/sensorSupply AT 303 : BOOL := true;
    pumpingTank2/extraction/pump/onCmd AT 306 : BOOL := false;
    pumpingTank2/extraction/pump/inputFlow AT 93 : REAL := 0.0;
    pumpingTank2/extraction/pump/onFB AT 308 : BOOL := false;
    pumpingTank2/extraction/pump/thermal AT 307 : BOOL := false;
    pumpingTank2/extraction/pump/speedVal AT 87 : REAL := 0.0;
    pumpingTank2/extraction/pump/outputFlow AT 91 : REAL := 0.0;
    pumpingTank2/extraction/pump/increment AT 116 : REAL := 0.0;
    pumpingTank2/extraction/pump/onState AT 315 : BOOL := false;
    pumpingTank2/extraction/pump/speedSetpoint AT 117 : REAL := 0.0;
    pumpingTank2/extraction/pump/unit AT 118 : REAL := 0.0;
    pumpingTank2/extraction/pump/nominalTime AT 119 : REAL := 2.0;
    pumpingTank2/extraction/pump/thermalLogic AT 316 : BOOL := false;
    pumpingTank2/extraction/pump/onFbLogic AT 317 : BOOL := true;
    pumpingTank2/extraction/pump/flowMax AT 120 : REAL := 1000.0;
    pumpingTank2/extraction/pump/nominalSpeed AT 121 : REAL := 3600.0;
    pumpingTank2/extraction/pump/flowPerHour AT 318 : BOOL := false;
    pumpingTank2/extraction/pump/flowPerMinute AT 319 : BOOL := true;
    pumpingTank2/extraction/pump/d_locking AT 320 : BOOL := false;
    pumpingTank2/extraction/pump/v_d_locking AT 122 : REAL := 0.0;
    pumpingTank2/extraction/pump/d_flow AT 321 : BOOL := false;
    pumpingTank2/extraction/pump/v_d_flow AT 123 : REAL := 0.0;
    pumpingTank2/extraction/pump/d_electrical AT 322 : BOOL := false;
    pumpingTank2/extraction/pump/v_d_electrical AT 323 : BOOL := false;
    pumpingTank2/extraction/pump/d_onFB AT 324 : BOOL := false;
    pumpingTank2/extraction/pump/v_d_onFB AT 325 : BOOL := false;
    pumpingTank2/extraction/cmdOfMotor/autoMode AT 28 : BOOL := false;
    pumpingTank2/extraction/cmdOfMotor/manualMode AT 29 : BOOL := false;
    pumpingTank2/extraction/cmdOfMotor/autoCmd AT 32 : BOOL := false;
    pumpingTank2/extraction/cmdOfMotor/thermalFB AT 307 : BOOL := false;
    pumpingTank2/extraction/cmdOfMotor/onFB AT 308 : BOOL := false;
    pumpingTank2/extraction/cmdOfMotor/onPB AT 309 : BOOL := false;
    pumpingTank2/extraction/cmdOfMotor/offPB AT 310 : BOOL := false;
    pumpingTank2/extraction/cmdOfMotor/acknowledgePB AT 10 : BOOL := false;
    pumpingTank2/extraction/cmdOfMotor/cmd AT 306 : BOOL := false;
    pumpingTank2/extraction/cmdOfMotor/generalFault AT 235 : BOOL := false;
    pumpingTank2/extraction/cmdOfMotor/actions/autoMode AT 28 : BOOL := false;
    pumpingTank2/extraction/cmdOfMotor/actions/manualMode AT 29 : BOOL := false;
    pumpingTank2/extraction/cmdOfMotor/actions/autoCmd AT 32 : BOOL := false;
    pumpingTank2/extraction/cmdOfMotor/actions/onPB AT 309 : BOOL := false;
    pumpingTank2/extraction/cmdOfMotor/actions/offPB AT 310 : BOOL := false;
    pumpingTank2/extraction/cmdOfMotor/actions/generalFault AT 235 : BOOL := false;
    pumpingTank2/extraction/cmdOfMotor/actions/cmd AT 306 : BOOL := false;
    pumpingTank2/extraction/cmdOfMotor/faults1/cmd AT 306 : BOOL := false;
    pumpingTank2/extraction/cmdOfMotor/faults1/thermalFB AT 307 : BOOL := false;
    pumpingTank2/extraction/cmdOfMotor/faults1/onFB AT 308 : BOOL := false;
    pumpingTank2/extraction/cmdOfMotor/faults1/acknowledgePB AT 10 : BOOL := false;
    pumpingTank2/extraction/cmdOfMotor/faults1/generalFault AT 235 : BOOL := false;
    pumpingTank2/extraction/cmdOfMotor/faults1/thermalFault AT 326 : BOOL := false;
    pumpingTank2/extraction/cmdOfMotor/faults1/onFBFault AT 327 : BOOL := false;
    pumpingTank2/levelScale/inputValue AT 93 : REAL := 0.0;
    pumpingTank2/levelScale/realValue AT 94 : REAL := 0.0;
    pumpingTank2/levelScale/dintValue AT 611 : DINT := 0;
    pumpingTank2/levelScale/intValue AT 610 : INT := 0;
    pumpingTank2/levelScale/a AT 124 : REAL := 0.0;
    pumpingTank2/levelScale/b AT 125 : REAL := 0.0;
    pumpingTank2/levelScale/k AT 126 : REAL := 0.0;
    pumpingTank2/levelScale/minInput AT 127 : REAL := 0.0;
    pumpingTank2/levelScale/maxInput AT 128 : REAL := 500.0;
    pumpingTank2/levelScale/minOutput AT 129 : REAL := 0.0;
    pumpingTank2/levelScale/maxOutput AT 130 : REAL := 100.0;
    pumpingTank2/levelScale/d_scale AT 330 : BOOL := false;
    pumpingTank2/levelScale/v_d_scale AT 131 : REAL := 0.0;
    pumpingTank2/highLevel/level AT 93 : REAL := 0.0;
    pumpingTank2/highLevel/sensorSupply AT 234 : BOOL := true;
    pumpingTank2/highLevel/thresholdSensor AT 13 : BOOL := false;
    pumpingTank2/highLevel/threshold AT 132 : REAL := 490.0;
    pumpingTank2/highLevel/wiringLogic AT 331 : BOOL := true;
    pumpingTank2/highLevel/d_sensor AT 332 : BOOL := false;
    pumpingTank2/highLevel/v_d_sensor AT 333 : BOOL := false;
    pumpingTank2/lowLevel/level AT 93 : REAL := 0.0;
    pumpingTank2/lowLevel/sensorSupply AT 233 : BOOL := true;
    pumpingTank2/lowLevel/thresholdSensor AT 14 : BOOL := false;
    pumpingTank2/lowLevel/threshold AT 133 : REAL := 30.0;
    pumpingTank2/lowLevel/wiringLogic AT 334 : BOOL := false;
    pumpingTank2/lowLevel/d_sensor AT 335 : BOOL := false;
    pumpingTank2/lowLevel/v_d_sensor AT 336 : BOOL := false;
    pumpingTank2/levelMeasurement/measure AT 94 : REAL := 0.0;
    pumpingTank2/levelMeasurement/sensorSupply AT 232 : BOOL := true;
    pumpingTank2/levelMeasurement/realValue AT 18 : REAL := 0.0;
    pumpingTank2/levelMeasurement/intValue AT 86 : REAL := 0.0;
    pumpingTank2/levelMeasurement/dintValue AT 85 : REAL := 0.0;
    pumpingTank2/levelMeasurement/tmp AT 684 : DINT := 0;
    pumpingTank2/levelMeasurement/localValue AT 134 : REAL := 0.0;
    pumpingTank2/levelMeasurement/nbDigit AT 685 : SINT := 2;
    pumpingTank2/levelMeasurement/d_value AT 337 : BOOL := false;
    pumpingTank2/levelMeasurement/v_d_value AT 135 : REAL := 0.0;
    flowsAdd/in1 AT 20 : REAL := 0.0;
    flowsAdd/in2 AT 21 : REAL := 0.0;
    flowsAdd/value AT 22 : REAL := 0.0;
    flowsAdd/dintValue AT 524 : DINT := 0;
    flowsAdd/intValue AT 523 : INT := 0;
    flowsAdd/d_locking AT 338 : BOOL := false;
    flowsAdd/v_d_locking AT 136 : REAL := 0.0;
    mixing/autoMode AT 28 : BOOL := false;
    mixing/manualMode AT 29 : BOOL := false;
    mixing/acknowledgePB AT 10 : BOOL := false;
    mixing/fillingValve AT 33 : BOOL := false;
    mixing/hiSpeedAgitator AT 34 : BOOL := false;
    mixing/loSpeedAgitator AT 35 : BOOL := false;
    mixing/inputFlow AT 22 : REAL := 0.0;
    mixing/highLevel AT 15 : BOOL := false;
    mixing/lowLevel AT 16 : BOOL := false;
    mixing/level AT 17 : REAL := 0.0;
    mixing/outputFlow AT 23 : REAL := 0.0;
    mixing/agitator/acknowledgePB AT 10 : BOOL := false;
    mixing/agitator/autoMode AT 28 : BOOL := false;
    mixing/agitator/manualMode AT 29 : BOOL := false;
    mixing/agitator/autoHSCmd AT 34 : BOOL := false;
    mixing/agitator/autoLSCmd AT 35 : BOOL := false;
    mixing/agitator/generalFault AT 345 : BOOL := false;
    mixing/agitator/speedVal AT 141 : REAL := 0.0;
    mixing/agitator/speedPercent AT 140 : REAL := 0.0;
    mixing/agitator/panel1/highSpeedPB AT 351 : BOOL := false;
    mixing/agitator/panel1/lowSpeedPB AT 352 : BOOL := false;
    mixing/agitator/panel1/stopPB AT 353 : BOOL := false;
    mixing/agitator/panel1/highSpeedPB/PB AT 351 : BOOL := false;
    mixing/agitator/panel1/highSpeedPB/action AT 357 : BOOL := false;
    mixing/agitator/panel1/highSpeedPB/timeCounter AT 145 : REAL := 0.0;
    mixing/agitator/panel1/highSpeedPB/pulseDuration AT 146 : REAL := 5.0;
    mixing/agitator/panel1/highSpeedPB/PBLogic AT 358 : BOOL := true;
    mixing/agitator/panel1/lowSpeedPB/PB AT 352 : BOOL := false;
    mixing/agitator/panel1/lowSpeedPB/action AT 359 : BOOL := false;
    mixing/agitator/panel1/lowSpeedPB/timeCounter AT 147 : REAL := 0.0;
    mixing/agitator/panel1/lowSpeedPB/pulseDuration AT 148 : REAL := 5.0;
    mixing/agitator/panel1/lowSpeedPB/PBLogic AT 360 : BOOL := true;
    mixing/agitator/panel1/stopPB/PB AT 353 : BOOL := false;
    mixing/agitator/panel1/stopPB/action AT 361 : BOOL := false;
    mixing/agitator/panel1/stopPB/timeCounter AT 149 : REAL := 0.0;
    mixing/agitator/panel1/stopPB/pulseDuration AT 150 : REAL := 5.0;
    mixing/agitator/panel1/stopPB/PBLogic AT 362 : BOOL := true;
    mixing/agitator/agitator/voltage380 AT 348 : BOOL := true;
    mixing/agitator/agitator/cmdSupply AT 347 : BOOL := true;
    mixing/agitator/agitator/sensorSupply AT 346 : BOOL := true;
    mixing/agitator/agitator/highSpeed AT 349 : BOOL := false;
    mixing/agitator/agitator/lowSpeed AT 350 : BOOL := false;
    mixing/agitator/agitator/highSpeedFB AT 354 : BOOL := false;
    mixing/agitator/agitator/lowSpeedFB AT 355 : BOOL := false;
    mixing/agitator/agitator/thermal AT 356 : BOOL := false;
    mixing/agitator/agitator/speedVal AT 141 : REAL := 0.0;
    mixing/agitator/agitator/speedPercent AT 140 : REAL := 0.0;
    mixing/agitator/agitator/increment AT 151 : REAL := 0.0;
    mixing/agitator/agitator/memoHighSpeed AT 363 : BOOL := false;
    mixing/agitator/agitator/memoLowSpeed AT 364 : BOOL := false;
    mixing/agitator/agitator/highSpeedState AT 365 : BOOL := false;
    mixing/agitator/agitator/lowSpeedState AT 366 : BOOL := false;
    mixing/agitator/agitator/speedSetpoint AT 152 : REAL := 0.0;
    mixing/agitator/agitator/cnt AT 688 : DINT := 0;
    mixing/agitator/agitator/flipflop AT 367 : BOOL := false;
    mixing/agitator/agitator/nominalTime AT 153 : REAL := 0.5;
    mixing/agitator/agitator/thermalLogic AT 368 : BOOL := false;
    mixing/agitator/agitator/highSpeedFbLogic AT 369 : BOOL := true;
    mixing/agitator/agitator/lowSpeedFbLogic AT 370 : BOOL := true;
    mixing/agitator/agitator/nominalLowSpeed AT 154 : REAL := 2500.0;
    mixing/agitator/agitator/nominalHighSpeed AT 155 : REAL := 5000.0;
    mixing/agitator/agitator/d_locking AT 371 : BOOL := false;
    mixing/agitator/agitator/v_d_locking AT 156 : REAL := 0.0;
    mixing/agitator/agitator/d_electrical AT 372 : BOOL := false;
    mixing/agitator/agitator/v_d_electrical AT 373 : BOOL := false;
    mixing/agitator/agitator/d_highSpeedFB AT 374 : BOOL := false;
    mixing/agitator/agitator/v_d_highSpeedFB AT 375 : BOOL := false;
    mixing/agitator/agitator/d_lowSpeedFB AT 376 : BOOL := false;
    mixing/agitator/agitator/v_d_lowSpeedFB AT 377 : BOOL := false;
    mixing/agitator/cmdOfMotor/autoMode AT 28 : BOOL := false;
    mixing/agitator/cmdOfMotor/manualMode AT 29 : BOOL := false;
    mixing/agitator/cmdOfMotor/autoHSCmd AT 34 : BOOL := false;
    mixing/agitator/cmdOfMotor/autoLSCmd AT 35 : BOOL := false;
    mixing/agitator/cmdOfMotor/highSpeedPB AT 351 : BOOL := false;
    mixing/agitator/cmdOfMotor/lowSpeedPB AT 352 : BOOL := false;
    mixing/agitator/cmdOfMotor/stopPB AT 353 : BOOL := false;
    mixing/agitator/cmdOfMotor/highSpeedFB AT 354 : BOOL := false;
    mixing/agitator/cmdOfMotor/lowSpeedFB AT 355 : BOOL := false;
    mixing/agitator/cmdOfMotor/thermalFB AT 356 : BOOL := false;
    mixing/agitator/cmdOfMotor/acknowledgePB AT 10 : BOOL := false;
    mixing/agitator/cmdOfMotor/highSpeedCmd AT 349 : BOOL := false;
    mixing/agitator/cmdOfMotor/lowSpeedCmd AT 350 : BOOL := false;
    mixing/agitator/cmdOfMotor/generalFault AT 345 : BOOL := false;
    mixing/agitator/cmdOfMotor/actions/autoMode AT 28 : BOOL := false;
    mixing/agitator/cmdOfMotor/actions/manualMode AT 29 : BOOL := false;
    mixing/agitator/cmdOfMotor/actions/autoHSCmd AT 34 : BOOL := false;
    mixing/agitator/cmdOfMotor/actions/autoLSCmd AT 35 : BOOL := false;
    mixing/agitator/cmdOfMotor/actions/highSpeedPB AT 351 : BOOL := false;
    mixing/agitator/cmdOfMotor/actions/lowSpeedPB AT 352 : BOOL := false;
    mixing/agitator/cmdOfMotor/actions/stopPB AT 353 : BOOL := false;
    mixing/agitator/cmdOfMotor/actions/generalFault AT 345 : BOOL := false;
    mixing/agitator/cmdOfMotor/actions/highSpeedCmd AT 349 : BOOL := false;
    mixing/agitator/cmdOfMotor/actions/lowSpeedCmd AT 350 : BOOL := false;
    mixing/agitator/cmdOfMotor/faults1/highSpeedCmd AT 349 : BOOL := false;
    mixing/agitator/cmdOfMotor/faults1/lowSpeedCmd AT 350 : BOOL := false;
    mixing/agitator/cmdOfMotor/faults1/highSpeedFB AT 354 : BOOL := false;
    mixing/agitator/cmdOfMotor/faults1/lowSpeedFB AT 355 : BOOL := false;
    mixing/agitator/cmdOfMotor/faults1/thermalFB AT 356 : BOOL := false;
    mixing/agitator/cmdOfMotor/faults1/acknowledgePB AT 10 : BOOL := false;
    mixing/agitator/cmdOfMotor/faults1/generalFault AT 345 : BOOL := false;
    mixing/agitator/cmdOfMotor/faults1/thermalFault AT 378 : BOOL := false;
    mixing/agitator/cmdOfMotor/faults1/highSpeedFBFault AT 379 : BOOL := false;
    mixing/agitator/cmdOfMotor/faults1/lowSpeedFBFault AT 380 : BOOL := false;
    mixing/flow/inputFlow AT 142 : REAL := 0.0;
    mixing/flow/outputFlow AT 143 : REAL := 0.0;
    mixing/flow/unit AT 157 : REAL := 0.0;
    mixing/flow/flowMax AT 158 : REAL := 2000.0;
    mixing/flow/flowPerHour AT 385 : BOOL := false;
    mixing/flow/flowPerMinute AT 386 : BOOL := true;
    mixing/valve5/acknowledgePB AT 10 : BOOL := false;
    mixing/valve5/autoMode AT 28 : BOOL := false;
    mixing/valve5/manualMode AT 29 : BOOL := false;
    mixing/valve5/autoOpenCmd AT 33 : BOOL := false;
    mixing/valve5/inputFlow AT 143 : REAL := 0.0;
    mixing/valve5/openedSensor AT 344 : BOOL := false;
    mixing/valve5/closedSensor AT 343 : BOOL := false;
    mixing/valve5/generalFault AT 342 : BOOL := false;
    mixing/valve5/outputFlow AT 23 : REAL := 0.0;
    mixing/valve5/percentOpening AT 139 : REAL := 0.0;
    mixing/valve5/panel1/openValvePB AT 390 : BOOL := false;
    mixing/valve5/panel1/switch/variable AT 390 : BOOL := false;
    mixing/valve5/panel1/switch/leftPosition AT 392 : BOOL := false;
    mixing/valve5/panel1/switch/rightPosition AT 393 : BOOL := false;
    mixing/valve5/cmdOfValve/autoMode AT 28 : BOOL := false;
    mixing/valve5/cmdOfValve/manualMode AT 29 : BOOL := false;
    mixing/valve5/cmdOfValve/autoOpenCmd AT 33 : BOOL := false;
    mixing/valve5/cmdOfValve/openValvePB AT 390 : BOOL := false;
    mixing/valve5/cmdOfValve/openedSensorFB AT 344 : BOOL := false;
    mixing/valve5/cmdOfValve/closedSensorFB AT 343 : BOOL := false;
    mixing/valve5/cmdOfValve/acknowledgePB AT 10 : BOOL := false;
    mixing/valve5/cmdOfValve/openCmd AT 391 : BOOL := false;
    mixing/valve5/cmdOfValve/generalFault AT 342 : BOOL := false;
    mixing/valve5/cmdOfValve/actions/autoMode AT 28 : BOOL := false;
    mixing/valve5/cmdOfValve/actions/manualMode AT 29 : BOOL := false;
    mixing/valve5/cmdOfValve/actions/autoOpenCmd AT 33 : BOOL := false;
    mixing/valve5/cmdOfValve/actions/openValvePB AT 390 : BOOL := false;
    mixing/valve5/cmdOfValve/actions/generalFault AT 342 : BOOL := false;
    mixing/valve5/cmdOfValve/actions/openCmd AT 391 : BOOL := false;
    mixing/valve5/cmdOfValve/faults1/openCmd AT 391 : BOOL := false;
    mixing/valve5/cmdOfValve/faults1/openedSensorFB AT 344 : BOOL := false;
    mixing/valve5/cmdOfValve/faults1/closedSensorFB AT 343 : BOOL := false;
    mixing/valve5/cmdOfValve/faults1/acknowledgePB AT 10 : BOOL := false;
    mixing/valve5/cmdOfValve/faults1/generalFault AT 342 : BOOL := false;
    mixing/valve5/cmdOfValve/faults1/discordanceFault AT 394 : BOOL := false;
    mixing/valve5/cmdOfValve/faults1/openedSensorFault AT 395 : BOOL := false;
    mixing/valve5/cmdOfValve/faults1/closedSensorFault AT 396 : BOOL := false;
    mixing/valve5/cmdOfValve/faults1/presetMvt AT 705 : TIME := T#0h0m4s0ms;
    mixing/valve5/cmdOfValve/faults1/presetDiscordance AT 709 : TIME := T#0h0m0s200ms;
    mixing/valve5/valve/voltage380 AT 389 : BOOL := true;
    mixing/valve5/valve/cmdSupply AT 388 : BOOL := true;
    mixing/valve5/valve/sensorSupply AT 387 : BOOL := true;
    mixing/valve5/valve/openCmd AT 391 : BOOL := false;
    mixing/valve5/valve/inputFlow AT 143 : REAL := 0.0;
    mixing/valve5/valve/openedSensor AT 344 : BOOL := false;
    mixing/valve5/valve/closedSensor AT 343 : BOOL := false;
    mixing/valve5/valve/outputFlow AT 23 : REAL := 0.0;
    mixing/valve5/valve/percentOpening AT 139 : REAL := 0.0;
    mixing/valve5/valve/increment AT 159 : REAL := 0.0;
    mixing/valve5/valve/openState AT 403 : BOOL := false;
    mixing/valve5/valve/closeState AT 404 : BOOL := false;
    mixing/valve5/valve/openingVal AT 160 : REAL := 0.0;
    mixing/valve5/valve/unit AT 161 : REAL := 0.0;
    mixing/valve5/valve/openingTime AT 162 : REAL := 2.0;
    mixing/valve5/valve/openedSensorLogic AT 405 : BOOL := true;
    mixing/valve5/valve/closedSensorLogic AT 406 : BOOL := true;
    mixing/valve5/valve/flowMax AT 163 : REAL := 100000.0;
    mixing/valve5/valve/flowPerHour AT 407 : BOOL := false;
    mixing/valve5/valve/flowPerMinute AT 408 : BOOL := false;
    mixing/valve5/valve/d_locking AT 409 : BOOL := false;
    mixing/valve5/valve/v_d_locking AT 164 : REAL := 0.0;
    mixing/valve5/valve/d_flow AT 410 : BOOL := false;
    mixing/valve5/valve/v_d_flow AT 165 : REAL := 0.0;
    mixing/valve5/valve/d_electrical AT 411 : BOOL := false;
    mixing/valve5/valve/v_d_electrical AT 412 : BOOL := false;
    mixing/valve5/valve/d_openedSensor AT 413 : BOOL := false;
    mixing/valve5/valve/v_d_openedSensor AT 414 : BOOL := false;
    mixing/valve5/valve/d_closedSensor AT 415 : BOOL := false;
    mixing/valve5/valve/v_d_closedSensor AT 416 : BOOL := false;
    mixing/mixingTank/inletFlow AT 22 : REAL := 0.0;
    mixing/mixingTank/outletFlow AT 23 : REAL := 0.0;
    mixing/mixingTank/tankLevel AT 142 : REAL := 0.0;
    mixing/mixingTank/percent AT 166 : REAL := 0.0;
    mixing/mixingTank/capacity AT 167 : REAL := 1000.0;
    mixing/mixingTank/d_level AT 417 : BOOL := false;
    mixing/mixingTank/v_d_level AT 168 : REAL := 0.0;
    mixing/levelScale/inputValue AT 142 : REAL := 0.0;
    mixing/levelScale/realValue AT 144 : REAL := 0.0;
    mixing/levelScale/dintValue AT 687 : DINT := 0;
    mixing/levelScale/intValue AT 686 : INT := 0;
    mixing/levelScale/a AT 169 : REAL := 0.0;
    mixing/levelScale/b AT 170 : REAL := 0.0;
    mixing/levelScale/k AT 171 : REAL := 0.0;
    mixing/levelScale/minInput AT 172 : REAL := 0.0;
    mixing/levelScale/maxInput AT 173 : REAL := 1000.0;
    mixing/levelScale/minOutput AT 174 : REAL := 0.0;
    mixing/levelScale/maxOutput AT 175 : REAL := 100.0;
    mixing/levelScale/d_scale AT 418 : BOOL := false;
    mixing/levelScale/v_d_scale AT 176 : REAL := 0.0;
    mixing/highLevel3/level AT 142 : REAL := 0.0;
    mixing/highLevel3/sensorSupply AT 341 : BOOL := true;
    mixing/highLevel3/thresholdSensor AT 15 : BOOL := false;
    mixing/highLevel3/threshold AT 177 : REAL := 950.0;
    mixing/highLevel3/wiringLogic AT 419 : BOOL := true;
    mixing/highLevel3/d_sensor AT 420 : BOOL := false;
    mixing/highLevel3/v_d_sensor AT 421 : BOOL := false;
    mixing/lowLevel3/level AT 142 : REAL := 0.0;
    mixing/lowLevel3/sensorSupply AT 340 : BOOL := true;
    mixing/lowLevel3/thresholdSensor AT 16 : BOOL := false;
    mixing/lowLevel3/threshold AT 178 : REAL := 100.0;
    mixing/lowLevel3/wiringLogic AT 422 : BOOL := false;
    mixing/lowLevel3/d_sensor AT 423 : BOOL := false;
    mixing/lowLevel3/v_d_sensor AT 424 : BOOL := false;
    mixing/levelMeasurement/measure AT 144 : REAL := 0.0;
    mixing/levelMeasurement/sensorSupply AT 339 : BOOL := true;
    mixing/levelMeasurement/realValue AT 17 : REAL := 0.0;
    mixing/levelMeasurement/intValue AT 138 : REAL := 0.0;
    mixing/levelMeasurement/dintValue AT 137 : REAL := 0.0;
    mixing/levelMeasurement/tmp AT 737 : DINT := 0;
    mixing/levelMeasurement/localValue AT 179 : REAL := 0.0;
    mixing/levelMeasurement/nbDigit AT 738 : SINT := 2;
    mixing/levelMeasurement/d_value AT 425 : BOOL := false;
    mixing/levelMeasurement/v_d_value AT 180 : REAL := 0.0;
    drive/autoMode AT 28 : BOOL := false;
    drive/manualMode AT 29 : BOOL := false;
    drive/acknowledgePB AT 10 : BOOL := false;
    drive/load AT 36 : BOOL := false;
    drive/evacuate AT 37 : BOOL := false;
    drive/convoy AT 38 : BOOL := false;
    drive/inputFlow AT 23 : REAL := 0.0;
    drive/bottlePresent AT 24 : BOOL := false;
    drive/bottleFilled AT 23 : BOOL := false;
    drive/pulse AT 22 : BOOL := false;
    drive/conveyor/autoMode AT 28 : BOOL := false;
    drive/conveyor/manualMode AT 29 : BOOL := false;
    drive/conveyor/autoCmd AT 38 : BOOL := false;
    drive/conveyor/acknowledgePB AT 10 : BOOL := false;
    drive/conveyor/speedVal AT 181 : REAL := 0.0;
    drive/conveyor/speedPercent AT 182 : REAL := 0.0;
    drive/conveyor/generalFault AT 427 : BOOL := false;
    drive/conveyor/panel1/forwardPB AT 434 : BOOL := false;
    drive/conveyor/panel1/stopPB AT 435 : BOOL := false;
    drive/conveyor/panel1/forwardPB/PB AT 434 : BOOL := false;
    drive/conveyor/panel1/forwardPB/action AT 436 : BOOL := false;
    drive/conveyor/panel1/forwardPB/timeCounter AT 183 : REAL := 0.0;
    drive/conveyor/panel1/forwardPB/pulseDuration AT 184 : REAL := 5.0;
    drive/conveyor/panel1/forwardPB/PBLogic AT 437 : BOOL := true;
    drive/conveyor/panel1/stopPB/PB AT 435 : BOOL := false;
    drive/conveyor/panel1/stopPB/action AT 438 : BOOL := false;
    drive/conveyor/panel1/stopPB/timeCounter AT 185 : REAL := 0.0;
    drive/conveyor/panel1/stopPB/pulseDuration AT 186 : REAL := 5.0;
    drive/conveyor/panel1/stopPB/PBLogic AT 439 : BOOL := true;
    drive/conveyor/motor/voltage380 AT 430 : BOOL := true;
    drive/conveyor/motor/cmdSupply AT 429 : BOOL := true;
    drive/conveyor/motor/sensorSupply AT 428 : BOOL := true;
    drive/conveyor/motor/forward AT 431 : BOOL := false;
    drive/conveyor/motor/forwardFB AT 432 : BOOL := false;
    drive/conveyor/motor/thermal AT 433 : BOOL := false;
    drive/conveyor/motor/speedVal AT 181 : REAL := 0.0;
    drive/conveyor/motor/speedPercent AT 182 : REAL := 0.0;
    drive/conveyor/motor/increment AT 187 : REAL := 0.0;
    drive/conveyor/motor/memoFwd AT 440 : BOOL := false;
    drive/conveyor/motor/forwardState AT 441 : BOOL := false;
    drive/conveyor/motor/wantedSpeed AT 188 : REAL := 0.0;
    drive/conveyor/motor/nominalSpeed AT 189 : REAL := 5000.0;
    drive/conveyor/motor/nominalTime AT 190 : REAL := 0.5;
    drive/conveyor/motor/thermalLogic AT 442 : BOOL := false;
    drive/conveyor/motor/feedbackLogic AT 443 : BOOL := true;
    drive/conveyor/motor/d_locking AT 444 : BOOL := false;
    drive/conveyor/motor/v_d_locking AT 191 : REAL := 0.0;
    drive/conveyor/motor/d_feedback AT 445 : BOOL := false;
    drive/conveyor/motor/v_d_feedback AT 446 : BOOL := false;
    drive/conveyor/motor/d_electrical AT 447 : BOOL := false;
    drive/conveyor/motor/v_d_electrical AT 448 : BOOL := false;
    drive/conveyor/cmdOfMotor/autoMode AT 28 : BOOL := false;
    drive/conveyor/cmdOfMotor/manualMode AT 29 : BOOL := false;
    drive/conveyor/cmdOfMotor/autoCmd AT 38 : BOOL := false;
    drive/conveyor/cmdOfMotor/forwardFB AT 432 : BOOL := false;
    drive/conveyor/cmdOfMotor/thermalFB AT 433 : BOOL := false;
    drive/conveyor/cmdOfMotor/forwardPB AT 434 : BOOL := false;
    drive/conveyor/cmdOfMotor/stopPB AT 435 : BOOL := false;
    drive/conveyor/cmdOfMotor/acknowledgePB AT 10 : BOOL := false;
    drive/conveyor/cmdOfMotor/forwardCmd AT 431 : BOOL := false;
    drive/conveyor/cmdOfMotor/generalFault AT 427 : BOOL := false;
    drive/conveyor/cmdOfMotor/actions/autoMode AT 28 : BOOL := false;
    drive/conveyor/cmdOfMotor/actions/manualMode AT 29 : BOOL := false;
    drive/conveyor/cmdOfMotor/actions/autoCmd AT 38 : BOOL := false;
    drive/conveyor/cmdOfMotor/actions/forwardPB AT 434 : BOOL := false;
    drive/conveyor/cmdOfMotor/actions/stopPB AT 435 : BOOL := false;
    drive/conveyor/cmdOfMotor/actions/generalFault AT 427 : BOOL := false;
    drive/conveyor/cmdOfMotor/actions/forwardCmd AT 431 : BOOL := false;
    drive/conveyor/cmdOfMotor/faults1/forwardCmd AT 431 : BOOL := false;
    drive/conveyor/cmdOfMotor/faults1/thermalFB AT 433 : BOOL := false;
    drive/conveyor/cmdOfMotor/faults1/forwardFB AT 432 : BOOL := false;
    drive/conveyor/cmdOfMotor/faults1/acknowledgePB AT 10 : BOOL := false;
    drive/conveyor/cmdOfMotor/faults1/generalFault AT 427 : BOOL := false;
    drive/conveyor/cmdOfMotor/faults1/thermalFault AT 449 : BOOL := false;
    drive/conveyor/cmdOfMotor/faults1/forwardFault AT 450 : BOOL := false;
    drive/pulse/speed AT 182 : REAL := 0.0;
    drive/pulse/sensorSupply AT 426 : BOOL := true;
    drive/pulse/pulseSensor AT 22 : BOOL := false;
    drive/pulse/counter AT 192 : REAL := 0.0;
    drive/pulse/pulseDuration AT 193 : REAL := 0.3;
    drive/pulse/d_sensor AT 453 : BOOL := false;
    drive/pulse/v_d_sensor AT 454 : BOOL := false;
    drive/bottles/pulseGenerator AT 22 : BOOL := false;
    drive/bottles/loading AT 36 : BOOL := false;
    drive/bottles/evacuation AT 37 : BOOL := false;
    drive/bottles/inputFlow AT 23 : REAL := 0.0;
    drive/bottles/bottleFilled AT 23 : BOOL := false;
    drive/bottles/bottlePresent AT 24 : BOOL := false;
    drive/bottles/existenceOfBottle1 AT 455 : BOOL := false;
    drive/bottles/existenceOfBottle2 AT 456 : BOOL := false;
    drive/bottles/existenceOfBottle3 AT 457 : BOOL := false;
    drive/bottles/levelOfBottle1 AT 194 : REAL := 0.0;
    drive/bottles/levelOfBottle2 AT 195 : REAL := 0.0;
    drive/bottles/levelOfBottle3 AT 196 : REAL := 0.0;
    drive/bottles/positionOfBottle1 AT 747 : DINT := 0;
    drive/bottles/positionOfBottle2 AT 748 : DINT := 0;
    drive/bottles/positionOfBottle3 AT 749 : DINT := 0;
    drive/bottles/edge_loading AT 458 : BOOL := false;
    drive/bottles/edge_evacuation AT 459 : BOOL := false;
    drive/bottles/edge_pulseGenerator AT 460 : BOOL := false;
    drive/bottles/first AT 461 : BOOL := true;
    drive/bottles/maxLevel AT 197 : REAL := 100.0;
    drive/bottles/increment AT 750 : INT := 1;
  END_VAR
END_CONFIGURATION
